LIN {X 0,Y 100.665,Z 312.75,A -85,B 0,C 180,E1 -26589.863,E2 -26589.863} C_VEL
LIN {X 0,Y 100.701,Z 312.753,A -85,B 0,C 180,E1 -26595.772,E2 -26595.772} C_VEL
LIN {X 0,Y 100.661,Z 312.753,A -85,B 0,C 180,E1 -26601.099,E2 -26601.099} C_VEL
LIN {X 0,Y 100.673,Z 312.753,A -85,B 0,C 180,E1 -26606.886,E2 -26606.886} C_VEL
LIN {X 0,Y 100.759,Z 312.744,A -85,B 0,C 180,E1 -26615.283,E2 -26615.283} C_VEL
LIN {X 0,Y 100.778,Z 312.74,A -85,B 0,C 180,E1 -26619.616,E2 -26619.616} C_VEL
LIN {X 0,Y 101.104,Z 312.698,A -85,B 0,C 180,E1 -26627.985,E2 -26627.985} C_VEL
LIN {X 0,Y 101.211,Z 312.69,A -85,B 0,C 180,E1 -26632.038,E2 -26632.038} C_VEL
LIN {X 0,Y 101.814,Z 312.615,A -85,B 0,C 180,E1 -26640.02,E2 -26640.02} C_VEL
LIN {X 0,Y 101.213,Z 312.689,A -85,B 0,C 180,E1 -26648.003,E2 -26648.003} C_VEL
LIN {X 0,Y 101.044,Z 312.702,A -85,B 0,C 180,E1 -26653.189,E2 -26653.189} C_VEL
LIN {X 0,Y 100.771,Z 312.742,A -85,B 0,C 180,E1 -26660.429,E2 -26660.429} C_VEL
LIN {X 0,Y 100.702,Z 312.75,A -85,B 0,C 180,E1 -26664.887,E2 -26664.887} C_VEL
LIN {X 0,Y 100.687,Z 312.75,A -85,B 0,C 180,E1 -26673.125,E2 -26673.125} C_VEL
LIN {X 0,Y 100.643,Z 312.753,A -85,B 0,C 180,E1 -26679.824,E2 -26679.824} C_VEL
LIN {X 0,Y 100.652,Z 312.76,A -85,B 0,C 180,E1 -26685.724,E2 -26685.724} C_VEL
LIN {X 0,Y 100.635,Z 312.757,A -85,B 0,C 180,E1 -26691.068,E2 -26691.068} C_VEL
LIN {X 0,Y 100.747,Z 312.743,A -85,B 0,C 180,E1 -26696.867,E2 -26696.867} C_VEL
LIN {X 0,Y 100.816,Z 312.737,A -85,B 0,C 180,E1 -26700.8,E2 -26700.8} C_VEL
LIN {X 0,Y 100.943,Z 312.723,A -85,B 0,C 180,E1 -26705.316,E2 -26705.316} C_VEL
LIN {X 0,Y 101.451,Z 312.659,A -85,B 0,C 180,E1 -26718.012,E2 -26718.012} C_VEL
LIN {X 0,Y 102.379,Z 312.611,A -85,B 0,C 180,E1 -26720.25,E2 -26720.25} C_VEL
LIN {X 0,Y 104.384,Z 336.262,A -85,B 0,C 180,E1 -26723.361,E2 -26723.361} C_VEL
LIN {X 0,Y 106.398,Z 352.42,A -85,B 0,C 180,E1 -26725.335,E2 -26725.335} C_VEL
LIN {X 0,Y 107.925,Z 383.014,A -85,B 0,C 180,E1 -26729.89,E2 -26729.89} C_VEL
LIN {X 0,Y 108.387,Z 393.278,A -85,B 0,C 180,E1 -26731.864,E2 -26731.864} C_VEL
LIN {X 0,Y 108.985,Z 404.094,A -85,B 0,C 180,E1 -26734.63,E2 -26734.63} C_VEL
LIN {X 0,Y 109.704,Z 414.44,A -85,B 0,C 180,E1 -26738.136,E2 -26738.136} C_VEL
LIN {X 0,Y 109.906,Z 418.538,A -85,B 0,C 180,E1 -26739.991,E2 -26739.991} C_VEL
LIN {X 0,Y 109.314,Z 424.896,A -85,B 0,C 180,E1 -26744.01,E2 -26744.01} C_VEL
LIN {X 0,Y 109.51,Z 433.596,A -85,B 0,C 180,E1 -26750.675,E2 -26750.675} C_VEL
LIN {X 0,Y 112.549,Z 441.833,A -85,B 0,C 180,E1 -26758.135,E2 -26758.135} C_VEL
LIN {X 0,Y 116.222,Z 446.661,A -85,B 0,C 180,E1 -26762.979,E2 -26762.979} C_VEL
LIN {X 0,Y 121.104,Z 450.868,A -85,B 0,C 180,E1 -26767.548,E2 -26767.548} C_VEL
LIN {X 0,Y 127.149,Z 454.377,A -85,B 0,C 180,E1 -26771.557,E2 -26771.557} C_VEL
LIN {X 0,Y 131.686,Z 456.416,A -85,B 0,C 180,E1 -26773.938,E2 -26773.938} C_VEL
LIN {X 0,Y 136.655,Z 458.059,A -85,B 0,C 180,E1 -26776.061,E2 -26776.061} C_VEL
LIN {X 0,Y 129.507,Z 454.575,A -85,B 0,C 180,E1 -26779.349,E2 -26779.349} C_VEL
LIN {X 0,Y 122.955,Z 450.261,A -85,B 0,C 180,E1 -26783.1,E2 -26783.1} C_VEL
LIN {X 0,Y 117.303,Z 444.969,A -85,B 0,C 180,E1 -26787.351,E2 -26787.351} C_VEL
LIN {X 0,Y 112.243,Z 437.819,A -85,B 0,C 180,E1 -26792.944,E2 -26792.944} C_VEL
LIN {X 0,Y 108.802,Z 428.944,A -85,B 0,C 180,E1 -26799.172,E2 -26799.172} C_VEL
LIN {X 0,Y 107.58,Z 421.613,A -85,B 0,C 180,E1 -26803.862,E2 -26803.862} C_VEL
LIN {X 0,Y 107.219,Z 414.624,A -85,B 0,C 180,E1 -26807.681,E2 -26807.681} C_VEL
LIN {X 0,Y 107.195,Z 406.282,A -85,B 0,C 180,E1 -26811.497,E2 -26811.497} C_VEL
LIN {X 0,Y 107.087,Z 396.993,A -85,B 0,C 180,E1 -26814.804,E2 -26814.804} C_VEL
LIN {X 0,Y 106.94,Z 388.426,A -85,B 0,C 180,E1 -26817.156,E2 -26817.156} C_VEL
LIN {X 0,Y 106.923,Z 378.584,A -85,B 0,C 180,E1 -26819.275,E2 -26819.275} C_VEL
LIN {X 0,Y 106.708,Z 365.006,A -85,B 0,C 180,E1 -26821.514,E2 -26821.514} C_VEL
LIN {X 0,Y 106.169,Z 353.16,A -85,B 0,C 180,E1 -26823.272,E2 -26823.272} C_VEL
LIN {X 0,Y 105.327,Z 347.436,A -85,B 0,C 180,E1 -26823.931,E2 -26823.931} C_VEL
LIN {X 0,Y 99.604,Z 328.593,A -85,B 0,C 180,E1 -26825.273,E2 -26825.273} C_VEL
LIN {X 0,Y 98.786,Z 322.861,A -85,B 0,C 180,E1 -26825.965,E2 -26825.965} C_VEL
LIN {X 0,Y 97.433,Z 313.16,A -85,B 0,C 180,E1 -26827.229,E2 -26827.229} C_VEL
LIN {X 0,Y 94.53,Z 313.52,A -85,B 0,C 180,E1 -26834.845,E2 -26834.845} C_VEL
LIN {X 0,Y 93.661,Z 313.629,A -85,B 0,C 180,E1 -26845.77,E2 -26845.77} C_VEL
LIN {X 0,Y 93.57,Z 313.64,A -85,B 0,C 180,E1 -26854.277,E2 -26854.277} C_VEL
LIN {X 0,Y 93.507,Z 313.646,A -85,B 0,C 180,E1 -26862.534,E2 -26862.534} C_VEL
LIN {X 0,Y 93.506,Z 313.642,A -85,B 0,C 180,E1 -26868.693,E2 -26868.693} C_VEL
LIN {X 0,Y 93.556,Z 313.642,A -85,B 0,C 180,E1 -26875.68,E2 -26875.68} C_VEL
LIN {X 0,Y 93.637,Z 313.633,A -85,B 0,C 180,E1 -26884.19,E2 -26884.19} C_VEL
LIN {X 0,Y 93.657,Z 313.623,A -85,B 0,C 180,E1 -26887.956,E2 -26887.956} C_VEL
LIN {X 0,Y 94.038,Z 313.575,A -85,B 0,C 180,E1 -26897.036,E2 -26897.036} C_VEL
LIN {X 0,Y 94.149,Z 313.57,A -85,B 0,C 180,E1 -26901.407,E2 -26901.407} C_VEL
LIN {X 0,Y 94.76,Z 313.495,A -85,B 0,C 180,E1 -26909.993,E2 -26909.993} C_VEL
LIN {X 0,Y 94.145,Z 313.571,A -85,B 0,C 180,E1 -26918.579,E2 -26918.579} C_VEL
LIN {X 0,Y 93.987,Z 313.581,A -85,B 0,C 180,E1 -26923.673,E2 -26923.673} C_VEL
LIN {X 0,Y 93.648,Z 313.624,A -85,B 0,C 180,E1 -26932.031,E2 -26932.031} C_VEL
LIN {X 0,Y 93.582,Z 313.641,A -85,B 0,C 180,E1 -26936.773,E2 -26936.773} C_VEL
LIN {X 0,Y 93.574,Z 313.639,A -85,B 0,C 180,E1 -26944.336,E2 -26944.336} C_VEL
LIN {X 0,Y 93.597,Z 313.635,A -85,B 0,C 180,E1 -26952.505,E2 -26952.505} C_VEL
LIN {X 0,Y 93.594,Z 313.632,A -85,B 0,C 180,E1 -26958.656,E2 -26958.656} C_VEL
LIN {X 0,Y 93.58,Z 313.639,A -85,B 0,C 180,E1 -26965.687,E2 -26965.687} C_VEL
LIN {X 0,Y 93.641,Z 313.632,A -85,B 0,C 180,E1 -26974.223,E2 -26974.223} C_VEL
LIN {X 0,Y 93.658,Z 313.623,A -85,B 0,C 180,E1 -26977.988,E2 -26977.988} C_VEL
LIN {X 0,Y 93.996,Z 313.581,A -85,B 0,C 180,E1 -26987.061,E2 -26987.061} C_VEL
LIN {X 0,Y 94.141,Z 313.571,A -85,B 0,C 180,E1 -26991.435,E2 -26991.435} C_VEL
LIN {X 0,Y 94.743,Z 313.496,A -85,B 0,C 180,E1 -27000.021,E2 -27000.021} C_VEL
LIN {X 0,Y 94.143,Z 313.571,A -85,B 0,C 180,E1 -27008.608,E2 -27008.608} C_VEL
LIN {X 0,Y 93.952,Z 313.585,A -85,B 0,C 180,E1 -27013.514,E2 -27013.514} C_VEL
LIN {X 0,Y 93.634,Z 313.625,A -85,B 0,C 180,E1 -27022.064,E2 -27022.064} C_VEL
LIN {X 0,Y 93.55,Z 313.644,A -85,B 0,C 180,E1 -27026.815,E2 -27026.815} C_VEL
LIN {X 0,Y 93.586,Z 313.638,A -85,B 0,C 180,E1 -27034.318,E2 -27034.318} C_VEL
LIN {X 0,Y 93.538,Z 313.643,A -85,B 0,C 180,E1 -27042.575,E2 -27042.575} C_VEL
LIN {X 0,Y 93.544,Z 313.638,A -85,B 0,C 180,E1 -27048.733,E2 -27048.733} C_VEL
LIN {X 0,Y 93.626,Z 313.634,A -85,B 0,C 180,E1 -27055.694,E2 -27055.694} C_VEL
LIN {X 0,Y 93.787,Z 313.615,A -85,B 0,C 180,E1 -27063.29,E2 -27063.29} C_VEL
LIN {X 0,Y 93.638,Z 313.628,A -85,B 0,C 180,E1 -27067.967,E2 -27067.967} C_VEL
LIN {X 0,Y 94.083,Z 313.573,A -85,B 0,C 180,E1 -27077.058,E2 -27077.058} C_VEL
LIN {X 0,Y 96.014,Z 313.336,A -85,B 0,C 180,E1 -27082.099,E2 -27082.099} C_VEL
LIN {X 0,Y 98.175,Z 336.207,A -85,B 0,C 180,E1 -27085.298,E2 -27085.298} C_VEL
LIN {X 0,Y 100.242,Z 351.555,A -85,B 0,C 180,E1 -27087.244,E2 -27087.244} C_VEL
LIN {X 0,Y 102.166,Z 383.219,A -85,B 0,C 180,E1 -27092.224,E2 -27092.224} C_VEL
LIN {X 0,Y 102.668,Z 392.712,A -85,B 0,C 180,E1 -27094.178,E2 -27094.178} C_VEL
LIN {X 0,Y 103.409,Z 402.496,A -85,B 0,C 180,E1 -27096.837,E2 -27096.837} C_VEL
LIN {X 0,Y 104.274,Z 412.028,A -85,B 0,C 180,E1 -27100.197,E2 -27100.197} C_VEL
LIN {X 0,Y 104.461,Z 415.18,A -85,B 0,C 180,E1 -27101.651,E2 -27101.651} C_VEL
LIN {X 0,Y 103.914,Z 421.503,A -85,B 0,C 180,E1 -27105.703,E2 -27105.703} C_VEL
LIN {X 0,Y 104.221,Z 429.208,A -85,B 0,C 180,E1 -27111.777,E2 -27111.777} C_VEL
LIN {X 0,Y 106.678,Z 437.042,A -85,B 0,C 180,E1 -27118.645,E2 -27118.645} C_VEL
LIN {X 0,Y 112.583,Z 444.916,A -85,B 0,C 180,E1 -27126.38,E2 -27126.38} C_VEL
LIN {X 0,Y 118.015,Z 449.228,A -85,B 0,C 180,E1 -27130.932,E2 -27130.932} C_VEL
LIN {X 0,Y 126.967,Z 453.986,A -85,B 0,C 180,E1 -27136.027,E2 -27136.027} C_VEL
LIN {X 0,Y 117.676,Z 447.719,A -85,B 0,C 180,E1 -27141.144,E2 -27141.144} C_VEL
LIN {X 0,Y 111.038,Z 440.965,A -85,B 0,C 180,E1 -27146.351,E2 -27146.351} C_VEL
LIN {X 0,Y 106.067,Z 432.912,A -85,B 0,C 180,E1 -27152.346,E2 -27152.346} C_VEL
LIN {X 0,Y 103.591,Z 426.177,A -85,B 0,C 180,E1 -27157.019,E2 -27157.019} C_VEL
LIN {X 0,Y 102.021,Z 416.844,A -85,B 0,C 180,E1 -27162.956,E2 -27162.956} C_VEL
LIN {X 0,Y 101.631,Z 408.488,A -85,B 0,C 180,E1 -27167.449,E2 -27167.449} C_VEL
LIN {X 0,Y 101.499,Z 400.712,A -85,B 0,C 180,E1 -27170.737,E2 -27170.737} C_VEL
LIN {X 0,Y 101.294,Z 390.735,A -85,B 0,C 180,E1 -27174.007,E2 -27174.007} C_VEL
LIN {X 0,Y 101.084,Z 379.599,A -85,B 0,C 180,E1 -27176.723,E2 -27176.723} C_VEL
LIN {X 0,Y 100.766,Z 365.78,A -85,B 0,C 180,E1 -27179.273,E2 -27179.273} C_VEL
LIN {X 0,Y 98.786,Z 322.861,A -85,B 0,C 180,E1 -27185.965,E2 -27185.965} C_VEL
LIN {X 0,Y 98.291,Z 320.434,A -85,B 0,C 180,E1 -27186.595,E2 -27186.595} C_VEL
LIN {X 0,Y 96.85,Z 317.92,A -85,B 0,C 180,E1 -27187.917,E2 -27187.917} C_VEL
LIN {X 0,Y 94.432,Z 315.841,A -85,B 0,C 180,E1 -27190.08,E2 -27190.08} C_VEL
LIN {X 0,Y 91.311,Z 314.68,A -85,B 0,C 180,E1 -27193.245,E2 -27193.245} C_VEL
LIN {X 0,Y 87.725,Z 314.403,A -85,B 0,C 180,E1 -27198.434,E2 -27198.434} C_VEL
LIN {X 0,Y 86.632,Z 314.494,A -85,B 0,C 180,E1 -27202.725,E2 -27202.725} C_VEL
LIN {X 0,Y 86.461,Z 314.525,A -85,B 0,C 180,E1 -27209.161,E2 -27209.161} C_VEL
LIN {X 0,Y 86.487,Z 314.524,A -85,B 0,C 180,E1 -27215.636,E2 -27215.636} C_VEL
LIN {X 0,Y 86.451,Z 314.526,A -85,B 0,C 180,E1 -27222.965,E2 -27222.965} C_VEL
LIN {X 0,Y 86.429,Z 314.522,A -85,B 0,C 180,E1 -27229.409,E2 -27229.409} C_VEL
LIN {X 0,Y 86.499,Z 314.521,A -85,B 0,C 180,E1 -27235.328,E2 -27235.328} C_VEL
LIN {X 0,Y 86.552,Z 314.517,A -85,B 0,C 180,E1 -27243.22,E2 -27243.22} C_VEL
LIN {X 0,Y 86.609,Z 314.508,A -85,B 0,C 180,E1 -27251.052,E2 -27251.052} C_VEL
LIN {X 0,Y 86.895,Z 314.464,A -85,B 0,C 180,E1 -27255.95,E2 -27255.95} C_VEL
LIN {X 0,Y 87.057,Z 314.453,A -85,B 0,C 180,E1 -27260.701,E2 -27260.701} C_VEL
LIN {X 0,Y 87.687,Z 314.376,A -85,B 0,C 180,E1 -27269.992,E2 -27269.992} C_VEL
LIN {X 0,Y 87.053,Z 314.453,A -85,B 0,C 180,E1 -27279.284,E2 -27279.284} C_VEL
LIN {X 0,Y 86.89,Z 314.465,A -85,B 0,C 180,E1 -27284.035,E2 -27284.035} C_VEL
LIN {X 0,Y 86.601,Z 314.509,A -85,B 0,C 180,E1 -27288.934,E2 -27288.934} C_VEL
LIN {X 0,Y 86.544,Z 314.518,A -85,B 0,C 180,E1 -27296.771,E2 -27296.771} C_VEL
LIN {X 0,Y 86.499,Z 314.523,A -85,B 0,C 180,E1 -27305.704,E2 -27305.704} C_VEL
LIN {X 0,Y 86.524,Z 314.517,A -85,B 0,C 180,E1 -27313.065,E2 -27313.065} C_VEL
LIN {X 0,Y 86.519,Z 314.511,A -85,B 0,C 180,E1 -27319.504,E2 -27319.504} C_VEL
LIN {X 0,Y 86.528,Z 314.518,A -85,B 0,C 180,E1 -27325.381,E2 -27325.381} C_VEL
LIN {X 0,Y 86.556,Z 314.516,A -85,B 0,C 180,E1 -27333.254,E2 -27333.254} C_VEL
LIN {X 0,Y 86.595,Z 314.51,A -85,B 0,C 180,E1 -27341.082,E2 -27341.082} C_VEL
LIN {X 0,Y 86.859,Z 314.469,A -85,B 0,C 180,E1 -27346.119,E2 -27346.119} C_VEL
LIN {X 0,Y 87.044,Z 314.455,A -85,B 0,C 180,E1 -27350.731,E2 -27350.731} C_VEL
LIN {X 0,Y 87.673,Z 314.377,A -85,B 0,C 180,E1 -27360.023,E2 -27360.023} C_VEL
LIN {X 0,Y 87.049,Z 314.454,A -85,B 0,C 180,E1 -27369.315,E2 -27369.315} C_VEL
LIN {X 0,Y 86.854,Z 314.47,A -85,B 0,C 180,E1 -27374.072,E2 -27374.072} C_VEL
LIN {X 0,Y 86.587,Z 314.511,A -85,B 0,C 180,E1 -27378.969,E2 -27378.969} C_VEL
LIN {X 0,Y 86.525,Z 314.519,A -85,B 0,C 180,E1 -27386.706,E2 -27386.706} C_VEL
LIN {X 0,Y 86.507,Z 314.523,A -85,B 0,C 180,E1 -27395.681,E2 -27395.681} C_VEL
LIN {X 0,Y 86.462,Z 314.525,A -85,B 0,C 180,E1 -27402.995,E2 -27402.995} C_VEL
LIN {X 0,Y 86.468,Z 314.518,A -85,B 0,C 180,E1 -27409.452,E2 -27409.452} C_VEL
LIN {X 0,Y 86.566,Z 314.514,A -85,B 0,C 180,E1 -27415.378,E2 -27415.378} C_VEL
LIN {X 0,Y 86.718,Z 314.495,A -85,B 0,C 180,E1 -27423.105,E2 -27423.105} C_VEL
LIN {X 0,Y 86.501,Z 314.523,A -85,B 0,C 180,E1 -27431.044,E2 -27431.044} C_VEL
LIN {X 0,Y 88.127,Z 314.318,A -85,B 0,C 180,E1 -27440.83,E2 -27440.83} C_VEL
LIN {X 0,Y 89.757,Z 314.11,A -85,B 0,C 180,E1 -27444.25,E2 -27444.25} C_VEL
LIN {X 0,Y 92.272,Z 337.546,A -85,B 0,C 180,E1 -27447.687,E2 -27447.687} C_VEL
LIN {X 0,Y 94.26,Z 351.179,A -85,B 0,C 180,E1 -27449.488,E2 -27449.488} C_VEL
LIN {X 0,Y 96.686,Z 382.911,A -85,B 0,C 180,E1 -27454.828,E2 -27454.828} C_VEL
LIN {X 0,Y 97.469,Z 393.635,A -85,B 0,C 180,E1 -27457.256,E2 -27457.256} C_VEL
LIN {X 0,Y 98.39,Z 403.722,A -85,B 0,C 180,E1 -27460.294,E2 -27460.294} C_VEL
LIN {X 0,Y 99.138,Z 410.816,A -85,B 0,C 180,E1 -27463.058,E2 -27463.058} C_VEL
LIN {X 0,Y 98.946,Z 414.824,A -85,B 0,C 180,E1 -27465.418,E2 -27465.418} C_VEL
LIN {X 0,Y 98.986,Z 423.465,A -85,B 0,C 180,E1 -27472.001,E2 -27472.001} C_VEL
LIN {X 0,Y 100.588,Z 430.572,A -85,B 0,C 180,E1 -27478.147,E2 -27478.147} C_VEL
LIN {X 0,Y 104.715,Z 437.975,A -85,B 0,C 180,E1 -27485.018,E2 -27485.018} C_VEL
LIN {X 0,Y 111.315,Z 444.509,A -85,B 0,C 180,E1 -27491.531,E2 -27491.531} C_VEL
LIN {X 0,Y 117.69,Z 448.827,A -85,B 0,C 180,E1 -27495.781,E2 -27495.781} C_VEL
LIN {X 0,Y 117.158,Z 448.434,A -85,B 0,C 180,E1 -27496.358,E2 -27496.358} C_VEL
LIN {X 0,Y 108.566,Z 440.736,A -85,B 0,C 180,E1 -27502.028,E2 -27502.028} C_VEL
LIN {X 0,Y 104.228,Z 435.253,A -85,B 0,C 180,E1 -27506.179,E2 -27506.179} C_VEL
LIN {X 0,Y 100.153,Z 427.508,A -85,B 0,C 180,E1 -27511.706,E2 -27511.706} C_VEL
LIN {X 0,Y 97.873,Z 420.23,A -85,B 0,C 180,E1 -27516.717,E2 -27516.717} C_VEL
LIN {X 0,Y 96.686,Z 410.847,A -85,B 0,C 180,E1 -27522.476,E2 -27522.476} C_VEL
LIN {X 0,Y 96.23,Z 401.198,A -85,B 0,C 180,E1 -27527.323,E2 -27527.323} C_VEL
LIN {X 0,Y 95.904,Z 392.21,A -85,B 0,C 180,E1 -27530.645,E2 -27530.645} C_VEL
LIN {X 0,Y 95.59,Z 380.07,A -85,B 0,C 180,E1 -27533.912,E2 -27533.912} C_VEL
LIN {X 0,Y 95.058,Z 365.316,A -85,B 0,C 180,E1 -27536.8,E2 -27536.8} C_VEL
LIN {X 0,Y 92.405,Z 320.941,A -85,B 0,C 180,E1 -27544.248,E2 -27544.248} C_VEL
LIN {X 0,Y 91.254,Z 313.926,A -85,B 0,C 180,E1 -27545.122,E2 -27545.122} C_VEL
LIN {X 0,Y 89.146,Z 314.195,A -85,B 0,C 180,E1 -27549.048,E2 -27549.048} C_VEL
LIN {X 0,Y 86.632,Z 314.494,A -85,B 0,C 180,E1 -27562.725,E2 -27562.725} C_VEL
LIN {X 0,Y 86.231,Z 314.554,A -85,B 0,C 180,E1 -27565.314,E2 -27565.314} C_VEL
LIN {X 0,Y 84.74,Z 314.743,A -85,B 0,C 180,E1 -27569.154,E2 -27569.154} C_VEL
LIN {X 0,Y 79.479,Z 315.389,A -85,B 0,C 180,E1 -27581.333,E2 -27581.333} C_VEL
LIN {X 0,Y 79.318,Z 315.412,A -85,B 0,C 180,E1 -27584.259,E2 -27584.259} C_VEL
LIN {X 0,Y 79.357,Z 315.411,A -85,B 0,C 180,E1 -27592.803,E2 -27592.803} C_VEL
LIN {X 0,Y 79.449,Z 315.4,A -85,B 0,C 180,E1 -27602.14,E2 -27602.14} C_VEL
LIN {X 0,Y 79.478,Z 315.392,A -85,B 0,C 180,E1 -27609.277,E2 -27609.277} C_VEL
LIN {X 0,Y 79.79,Z 315.35,A -85,B 0,C 180,E1 -27615.557,E2 -27615.557} C_VEL
LIN {X 0,Y 79.937,Z 315.339,A -85,B 0,C 180,E1 -27619.864,E2 -27619.864} C_VEL
LIN {X 0,Y 80.614,Z 315.257,A -85,B 0,C 180,E1 -27629.992,E2 -27629.992} C_VEL
LIN {X 0,Y 79.933,Z 315.34,A -85,B 0,C 180,E1 -27640.119,E2 -27640.119} C_VEL
LIN {X 0,Y 79.702,Z 315.364,A -85,B 0,C 180,E1 -27645.33,E2 -27645.33} C_VEL
LIN {X 0,Y 79.469,Z 315.393,A -85,B 0,C 180,E1 -27650.707,E2 -27650.707} C_VEL
LIN {X 0,Y 79.443,Z 315.401,A -85,B 0,C 180,E1 -27657.852,E2 -27657.852} C_VEL
LIN {X 0,Y 79.415,Z 315.404,A -85,B 0,C 180,E1 -27667.251,E2 -27667.251} C_VEL
LIN {X 0,Y 79.432,Z 315.404,A -85,B 0,C 180,E1 -27675.046,E2 -27675.046} C_VEL
LIN {X 0,Y 79.419,Z 315.403,A -85,B 0,C 180,E1 -27682.775,E2 -27682.775} C_VEL
LIN {X 0,Y 79.454,Z 315.401,A -85,B 0,C 180,E1 -27692.175,E2 -27692.175} C_VEL
LIN {X 0,Y 79.472,Z 315.393,A -85,B 0,C 180,E1 -27699.313,E2 -27699.313} C_VEL
LIN {X 0,Y 79.761,Z 315.354,A -85,B 0,C 180,E1 -27705.716,E2 -27705.716} C_VEL
LIN {X 0,Y 79.922,Z 315.341,A -85,B 0,C 180,E1 -27709.897,E2 -27709.897} C_VEL
LIN {X 0,Y 80.603,Z 315.257,A -85,B 0,C 180,E1 -27720.025,E2 -27720.025} C_VEL
LIN {X 0,Y 79.925,Z 315.341,A -85,B 0,C 180,E1 -27730.154,E2 -27730.154} C_VEL
LIN {X 0,Y 79.682,Z 315.367,A -85,B 0,C 180,E1 -27735.369,E2 -27735.369} C_VEL
LIN {X 0,Y 79.459,Z 315.394,A -85,B 0,C 180,E1 -27740.745,E2 -27740.745} C_VEL
LIN {X 0,Y 79.421,Z 315.404,A -85,B 0,C 180,E1 -27747.781,E2 -27747.781} C_VEL
LIN {X 0,Y 79.345,Z 315.405,A -85,B 0,C 180,E1 -27752.131,E2 -27752.131} C_VEL
LIN {X 0,Y 79.37,Z 315.407,A -85,B 0,C 180,E1 -27758.334,E2 -27758.334} C_VEL
LIN {X 0,Y 79.395,Z 315.408,A -85,B 0,C 180,E1 -27765.118,E2 -27765.118} C_VEL
LIN {X 0,Y 79.409,Z 315.405,A -85,B 0,C 180,E1 -27772.839,E2 -27772.839} C_VEL
LIN {X 0,Y 79.621,Z 315.379,A -85,B 0,C 180,E1 -27782.016,E2 -27782.016} C_VEL
LIN {X 0,Y 79.45,Z 315.398,A -85,B 0,C 180,E1 -27789.288,E2 -27789.288} C_VEL
LIN {X 0,Y 80.661,Z 315.247,A -85,B 0,C 180,E1 -27799.973,E2 -27799.973} C_VEL
LIN {X 0,Y 83.808,Z 314.862,A -85,B 0,C 180,E1 -27806.885,E2 -27806.885} C_VEL
LIN {X 0,Y 86.75,Z 338.79,A -85,B 0,C 180,E1 -27810.516,E2 -27810.516} C_VEL
LIN {X 0,Y 88.662,Z 351.424,A -85,B 0,C 180,E1 -27812.279,E2 -27812.279} C_VEL
LIN {X 0,Y 91.375,Z 381.665,A -85,B 0,C 180,E1 -27817.604,E2 -27817.604} C_VEL
LIN {X 0,Y 92.214,Z 391.506,A -85,B 0,C 180,E1 -27819.881,E2 -27819.881} C_VEL
LIN {X 0,Y 93.145,Z 400.297,A -85,B 0,C 180,E1 -27822.536,E2 -27822.536} C_VEL
LIN {X 0,Y 94.053,Z 407.162,A -85,B 0,C 180,E1 -27825.168,E2 -27825.168} C_VEL
LIN {X 0,Y 94.054,Z 410.92,A -85,B 0,C 180,E1 -27827.398,E2 -27827.398} C_VEL
LIN {X 0,Y 94.378,Z 420.929,A -85,B 0,C 180,E1 -27835.213,E2 -27835.213} C_VEL
LIN {X 0,Y 97.286,Z 429.392,A -85,B 0,C 180,E1 -27842.814,E2 -27842.814} C_VEL
LIN {X 0,Y 101.408,Z 435.563,A -85,B 0,C 180,E1 -27848.597,E2 -27848.597} C_VEL
LIN {X 0,Y 108.867,Z 442.529,A -85,B 0,C 180,E1 -27855.252,E2 -27855.252} C_VEL
LIN {X 0,Y 107.666,Z 441.279,A -85,B 0,C 180,E1 -27856.965,E2 -27856.965} C_VEL
LIN {X 0,Y 100.944,Z 433.671,A -85,B 0,C 180,E1 -27862.446,E2 -27862.446} C_VEL
LIN {X 0,Y 96.984,Z 427.318,A -85,B 0,C 180,E1 -27867.056,E2 -27867.056} C_VEL
LIN {X 0,Y 93.114,Z 416.885,A -85,B 0,C 180,E1 -27874.282,E2 -27874.282} C_VEL
LIN {X 0,Y 91.723,Z 407.604,A -85,B 0,C 180,E1 -27880.1,E2 -27880.1} C_VEL
LIN {X 0,Y 91.279,Z 399.872,A -85,B 0,C 180,E1 -27884.112,E2 -27884.112} C_VEL
LIN {X 0,Y 90.791,Z 390.821,A -85,B 0,C 180,E1 -27887.687,E2 -27887.687} C_VEL
LIN {X 0,Y 90.263,Z 379.883,A -85,B 0,C 180,E1 -27890.878,E2 -27890.878} C_VEL
LIN {X 0,Y 89.58,Z 365.368,A -85,B 0,C 180,E1 -27893.926,E2 -27893.926} C_VEL
LIN {X 0,Y 86.423,Z 321.198,A -85,B 0,C 180,E1 -27901.797,E2 -27901.797} C_VEL
LIN {X 0,Y 85.244,Z 314.674,A -85,B 0,C 180,E1 -27902.708,E2 -27902.708} C_VEL
LIN {X 0,Y 83.804,Z 314.852,A -85,B 0,C 180,E1 -27904.786,E2 -27904.786} C_VEL
LIN {X 0,Y 79.565,Z 315.373,A -85,B 0,C 180,E1 -27922.535,E2 -27922.535} C_VEL
LIN {X 0,Y 79.471,Z 315.398,A -85,B 0,C 180,E1 -27927.812,E2 -27927.812} C_VEL
LIN {X 0,Y 79.367,Z 315.41,A -85,B 0,C 180,E1 -27937.147,E2 -27937.147} C_VEL
LIN {X 0,Y 79.318,Z 315.412,A -85,B 0,C 180,E1 -27944.259,E2 -27944.259} C_VEL
LIN {X 0,Y 79.152,Z 315.453,A -85,B 0,C 180,E1 -27947.087,E2 -27947.087} C_VEL
LIN {X 0,Y 77.932,Z 315.621,A -85,B 0,C 180,E1 -27951.302,E2 -27951.302} C_VEL
LIN {X 0,Y 74.763,Z 316.01,A -85,B 0,C 180,E1 -27958.483,E2 -27958.483} C_VEL
LIN {X 0,Y 72.708,Z 316.241,A -85,B 0,C 180,E1 -27964.68,E2 -27964.68} C_VEL
LIN {X 0,Y 72.339,Z 316.273,A -85,B 0,C 180,E1 -27967.914,E2 -27967.914} C_VEL
LIN {X 0,Y 72.686,Z 316.236,A -85,B 0,C 180,E1 -27975.095,E2 -27975.095} C_VEL
LIN {X 0,Y 72.827,Z 316.223,A -85,B 0,C 180,E1 -27978.862,E2 -27978.862} C_VEL
LIN {X 0,Y 73.54,Z 316.138,A -85,B 0,C 180,E1 -27989.991,E2 -27989.991} C_VEL
LIN {X 0,Y 72.822,Z 316.224,A -85,B 0,C 180,E1 -28001.119,E2 -28001.119} C_VEL
LIN {X 0,Y 72.532,Z 316.262,A -85,B 0,C 180,E1 -28006.889,E2 -28006.889} C_VEL
LIN {X 0,Y 72.352,Z 316.276,A -85,B 0,C 180,E1 -28012.854,E2 -28012.854} C_VEL
LIN {X 0,Y 72.337,Z 316.283,A -85,B 0,C 180,E1 -28019.089,E2 -28019.089} C_VEL
LIN {X 0,Y 72.3,Z 316.292,A -85,B 0,C 180,E1 -28025.666,E2 -28025.666} C_VEL
LIN {X 0,Y 72.276,Z 316.291,A -85,B 0,C 180,E1 -28032.882,E2 -28032.882} C_VEL
LIN {X 0,Y 72.326,Z 316.282,A -85,B 0,C 180,E1 -28041.005,E2 -28041.005} C_VEL
LIN {X 0,Y 72.305,Z 316.291,A -85,B 0,C 180,E1 -28044.361,E2 -28044.361} C_VEL
LIN {X 0,Y 72.363,Z 316.281,A -85,B 0,C 180,E1 -28050.982,E2 -28050.982} C_VEL
LIN {X 0,Y 72.359,Z 316.275,A -85,B 0,C 180,E1 -28057.17,E2 -28057.17} C_VEL
LIN {X 0,Y 72.658,Z 316.239,A -85,B 0,C 180,E1 -28065.261,E2 -28065.261} C_VEL
LIN {X 0,Y 72.809,Z 316.225,A -85,B 0,C 180,E1 -28068.898,E2 -28068.898} C_VEL
LIN {X 0,Y 73.531,Z 316.138,A -85,B 0,C 180,E1 -28080.028,E2 -28080.028} C_VEL
LIN {X 0,Y 72.818,Z 316.223,A -85,B 0,C 180,E1 -28091.157,E2 -28091.157} C_VEL
LIN {X 0,Y 72.497,Z 316.266,A -85,B 0,C 180,E1 -28096.936,E2 -28096.936} C_VEL
LIN {X 0,Y 72.344,Z 316.276,A -85,B 0,C 180,E1 -28102.895,E2 -28102.895} C_VEL
LIN {X 0,Y 72.315,Z 316.286,A -85,B 0,C 180,E1 -28109.103,E2 -28109.103} C_VEL
LIN {X 0,Y 72.289,Z 316.293,A -85,B 0,C 180,E1 -28115.717,E2 -28115.717} C_VEL
LIN {X 0,Y 72.254,Z 316.294,A -85,B 0,C 180,E1 -28122.947,E2 -28122.947} C_VEL
LIN {X 0,Y 72.311,Z 316.284,A -85,B 0,C 180,E1 -28131.075,E2 -28131.075} C_VEL
LIN {X 0,Y 72.483,Z 316.265,A -85,B 0,C 180,E1 -28140.818,E2 -28140.818} C_VEL
LIN {X 0,Y 72.401,Z 316.271,A -85,B 0,C 180,E1 -28147.163,E2 -28147.163} C_VEL
LIN {X 0,Y 75.084,Z 315.939,A -85,B 0,C 180,E1 -28164.638,E2 -28164.638} C_VEL
LIN {X 0,Y 78.13,Z 315.681,A -85,B 0,C 180,E1 -28169.929,E2 -28169.929} C_VEL
LIN {X 0,Y 81.078,Z 337.742,A -85,B 0,C 180,E1 -28173.425,E2 -28173.425} C_VEL
LIN {X 0,Y 83.185,Z 350.295,A -85,B 0,C 180,E1 -28175.189,E2 -28175.189} C_VEL
LIN {X 0,Y 86.499,Z 381.584,A -85,B 0,C 180,E1 -28180.986,E2 -28180.986} C_VEL
LIN {X 0,Y 87.533,Z 391.069,A -85,B 0,C 180,E1 -28183.354,E2 -28183.354} C_VEL
LIN {X 0,Y 88.702,Z 399.582,A -85,B 0,C 180,E1 -28186.107,E2 -28186.107} C_VEL
LIN {X 0,Y 89.448,Z 405.007,A -85,B 0,C 180,E1 -28188.325,E2 -28188.325} C_VEL
LIN {X 0,Y 89.402,Z 412.899,A -85,B 0,C 180,E1 -28194.229,E2 -28194.229} C_VEL
LIN {X 0,Y 91.666,Z 422.307,A -85,B 0,C 180,E1 -28202.467,E2 -28202.467} C_VEL
LIN {X 0,Y 94.686,Z 428.096,A -85,B 0,C 180,E1 -28207.768,E2 -28207.768} C_VEL
LIN {X 0,Y 100.628,Z 435.105,A -85,B 0,C 180,E1 -28214.308,E2 -28214.308} C_VEL
LIN {X 0,Y 101.188,Z 435.575,A -85,B 0,C 180,E1 -28215.984,E2 -28215.984} C_VEL
LIN {X 0,Y 94.574,Z 426.864,A -85,B 0,C 180,E1 -28222.163,E2 -28222.163} C_VEL
LIN {X 0,Y 90.096,Z 417.876,A -85,B 0,C 180,E1 -28228.468,E2 -28228.468} C_VEL
LIN {X 0,Y 87.575,Z 407.545,A -85,B 0,C 180,E1 -28235.344,E2 -28235.344} C_VEL
LIN {X 0,Y 86.666,Z 398.916,A -85,B 0,C 180,E1 -28240.304,E2 -28240.304} C_VEL
LIN {X 0,Y 86.178,Z 391.955,A -85,B 0,C 180,E1 -28243.392,E2 -28243.392} C_VEL
LIN {X 0,Y 85.544,Z 381.767,A -85,B 0,C 180,E1 -28246.768,E2 -28246.768} C_VEL
LIN {X 0,Y 84.757,Z 368.523,A -85,B 0,C 180,E1 -28249.978,E2 -28249.978} C_VEL
LIN {X 0,Y 81.023,Z 327.502,A -85,B 0,C 180,E1 -28257.8,E2 -28257.8} C_VEL
LIN {X 0,Y 80.22,Z 319.12,A -85,B 0,C 180,E1 -28259.269,E2 -28259.269} C_VEL
LIN {X 0,Y 79.558,Z 315.388,A -85,B 0,C 180,E1 -28259.816,E2 -28259.816} C_VEL
LIN {X 0,Y 77.405,Z 315.65,A -85,B 0,C 180,E1 -28262.712,E2 -28262.712} C_VEL
LIN {X 0,Y 72.503,Z 316.257,A -85,B 0,C 180,E1 -28282.782,E2 -28282.782} C_VEL
LIN {X 0,Y 72.349,Z 316.283,A -85,B 0,C 180,E1 -28289.025,E2 -28289.025} C_VEL
LIN {X 0,Y 72.277,Z 316.294,A -85,B 0,C 180,E1 -28295.655,E2 -28295.655} C_VEL
LIN {X 0,Y 72.226,Z 316.297,A -85,B 0,C 180,E1 -28302.892,E2 -28302.892} C_VEL
LIN {X 0,Y 72.267,Z 316.289,A -85,B 0,C 180,E1 -28311.03,E2 -28311.03} C_VEL
LIN {X 0,Y 72.265,Z 316.296,A -85,B 0,C 180,E1 -28314.29,E2 -28314.29} C_VEL
LIN {X 0,Y 72.329,Z 316.284,A -85,B 0,C 180,E1 -28320.923,E2 -28320.923} C_VEL
LIN {X 0,Y 72.339,Z 316.273,A -85,B 0,C 180,E1 -28327.914,E2 -28327.914} C_VEL
LIN {X 0,Y 71.739,Z 316.361,A -85,B 0,C 180,E1 -28332.596,E2 -28332.596} C_VEL
LIN {X 0,Y 69.917,Z 316.588,A -85,B 0,C 180,E1 -28338.848,E2 -28338.848} C_VEL
LIN {X 0,Y 65.999,Z 317.061,A -85,B 0,C 180,E1 -28353.987,E2 -28353.987} C_VEL
LIN {X 0,Y 65.716,Z 317.103,A -85,B 0,C 180,E1 -28362.34,E2 -28362.34} C_VEL
LIN {X 0,Y 65.338,Z 317.158,A -85,B 0,C 180,E1 -28368.814,E2 -28368.814} C_VEL
LIN {X 0,Y 65.206,Z 317.174,A -85,B 0,C 180,E1 -28375.527,E2 -28375.527} C_VEL
LIN {X 0,Y 65.176,Z 317.17,A -85,B 0,C 180,E1 -28382.613,E2 -28382.613} C_VEL
LIN {X 0,Y 65.212,Z 317.165,A -85,B 0,C 180,E1 -28391.078,E2 -28391.078} C_VEL
LIN {X 0,Y 65.233,Z 317.162,A -85,B 0,C 180,E1 -28399.771,E2 -28399.771} C_VEL
LIN {X 0,Y 65.23,Z 317.163,A -85,B 0,C 180,E1 -28409.512,E2 -28409.512} C_VEL
LIN {X 0,Y 65.215,Z 317.172,A -85,B 0,C 180,E1 -28414.501,E2 -28414.501} C_VEL
LIN {X 0,Y 65.568,Z 317.124,A -85,B 0,C 180,E1 -28424.684,E2 -28424.684} C_VEL
LIN {X 0,Y 65.702,Z 317.105,A -85,B 0,C 180,E1 -28427.679,E2 -28427.679} C_VEL
LIN {X 0,Y 66.429,Z 317.023,A -85,B 0,C 180,E1 -28440.03,E2 -28440.03} C_VEL
LIN {X 0,Y 65.713,Z 317.103,A -85,B 0,C 180,E1 -28452.382,E2 -28452.382} C_VEL
LIN {X 0,Y 65.325,Z 317.16,A -85,B 0,C 180,E1 -28458.861,E2 -28458.861} C_VEL
LIN {X 0,Y 65.188,Z 317.176,A -85,B 0,C 180,E1 -28465.579,E2 -28465.579} C_VEL
LIN {X 0,Y 65.155,Z 317.173,A -85,B 0,C 180,E1 -28472.673,E2 -28472.673} C_VEL
LIN {X 0,Y 65.188,Z 317.167,A -85,B 0,C 180,E1 -28481.019,E2 -28481.019} C_VEL
LIN {X 0,Y 65.217,Z 317.164,A -85,B 0,C 180,E1 -28489.73,E2 -28489.73} C_VEL
LIN {X 0,Y 65.333,Z 317.15,A -85,B 0,C 180,E1 -28499.436,E2 -28499.436} C_VEL
LIN {X 0,Y 65.296,Z 317.163,A -85,B 0,C 180,E1 -28504.511,E2 -28504.511} C_VEL
LIN {X 0,Y 67.535,Z 316.879,A -85,B 0,C 180,E1 -28524.037,E2 -28524.037} C_VEL
LIN {X 0,Y 72.103,Z 316.311,A -85,B 0,C 180,E1 -28532.803,E2 -28532.803} C_VEL
LIN {X 0,Y 72.727,Z 316.282,A -85,B 0,C 180,E1 -28533.472,E2 -28533.472} C_VEL
LIN {X 0,Y 76.015,Z 338.211,A -85,B 0,C 180,E1 -28537.064,E2 -28537.064} C_VEL
LIN {X 0,Y 78.285,Z 350.926,A -85,B 0,C 180,E1 -28538.916,E2 -28538.916} C_VEL
LIN {X 0,Y 82.132,Z 381.54,A -85,B 0,C 180,E1 -28544.883,E2 -28544.883} C_VEL
LIN {X 0,Y 83.53,Z 392.164,A -85,B 0,C 180,E1 -28547.766,E2 -28547.766} C_VEL
LIN {X 0,Y 84.818,Z 400.11,A -85,B 0,C 180,E1 -28550.627,E2 -28550.627} C_VEL
LIN {X 0,Y 85.043,Z 402.447,A -85,B 0,C 180,E1 -28551.84,E2 -28551.84} C_VEL
LIN {X 0,Y 85.764,Z 411.779,A -85,B 0,C 180,E1 -28559.459,E2 -28559.459} C_VEL
LIN {X 0,Y 88.583,Z 419.966,A -85,B 0,C 180,E1 -28566.807,E2 -28566.807} C_VEL
LIN {X 0,Y 92.932,Z 426.616,A -85,B 0,C 180,E1 -28572.902,E2 -28572.902} C_VEL
LIN {X 0,Y 94.412,Z 428.311,A -85,B 0,C 180,E1 -28575.623,E2 -28575.623} C_VEL
LIN {X 0,Y 89.322,Z 420.629,A -85,B 0,C 180,E1 -28580.964,E2 -28580.964} C_VEL
LIN {X 0,Y 84.767,Z 410.05,A -85,B 0,C 180,E1 -28588.332,E2 -28588.332} C_VEL
LIN {X 0,Y 82.848,Z 399.795,A -85,B 0,C 180,E1 -28594.878,E2 -28594.878} C_VEL
LIN {X 0,Y 82.076,Z 392.704,A -85,B 0,C 180,E1 -28598.634,E2 -28598.634} C_VEL
LIN {X 0,Y 81.356,Z 385.37,A -85,B 0,C 180,E1 -28601.575,E2 -28601.575} C_VEL
LIN {X 0,Y 80.486,Z 373.425,A -85,B 0,C 180,E1 -28604.967,E2 -28604.967} C_VEL
LIN {X 0,Y 79.29,Z 360.964,A -85,B 0,C 180,E1 -28607.725,E2 -28607.725} C_VEL
LIN {X 0,Y 74.966,Z 320.489,A -85,B 0,C 180,E1 -28615.773,E2 -28615.773} C_VEL
LIN {X 0,Y 74.158,Z 316.056,A -85,B 0,C 180,E1 -28616.407,E2 -28616.407} C_VEL
LIN {X 0,Y 70.322,Z 316.536,A -85,B 0,C 180,E1 -28621.718,E2 -28621.718} C_VEL
LIN {X 0,Y 65.709,Z 317.112,A -85,B 0,C 180,E1 -28638.682,E2 -28638.682} C_VEL
LIN {X 0,Y 65.214,Z 317.165,A -85,B 0,C 180,E1 -28650.423,E2 -28650.423} C_VEL
LIN {X 0,Y 65.161,Z 317.171,A -85,B 0,C 180,E1 -28660.961,E2 -28660.961} C_VEL
LIN {X 0,Y 65.176,Z 317.169,A -85,B 0,C 180,E1 -28669.672,E2 -28669.672} C_VEL
LIN {X 0,Y 65.196,Z 317.167,A -85,B 0,C 180,E1 -28679.518,E2 -28679.518} C_VEL
LIN {X 0,Y 65.166,Z 317.165,A -85,B 0,C 180,E1 -28688.047,E2 -28688.047} C_VEL
LIN {X 0,Y 65.583,Z 317.122,A -85,B 0,C 180,E1 -28694.551,E2 -28694.551} C_VEL
LIN {X 0,Y 65.722,Z 317.102,A -85,B 0,C 180,E1 -28697.64,E2 -28697.64} C_VEL
LIN {X 0,Y 66.463,Z 317.019,A -85,B 0,C 180,E1 -28709.99,E2 -28709.99} C_VEL
LIN {X 0,Y 65.999,Z 317.061,A -85,B 0,C 180,E1 -28713.987,E2 -28713.987} C_VEL
LIN {X 0,Y 65.05,Z 317.195,A -85,B 0,C 180,E1 -28719.083,E2 -28719.083} C_VEL
LIN {X 0,Y 63.349,Z 317.409,A -85,B 0,C 180,E1 -28724.174,E2 -28724.174} C_VEL
LIN {X 0,Y 59.486,Z 317.89,A -85,B 0,C 180,E1 -28734.963,E2 -28734.963} C_VEL
LIN {X 0,Y 58.099,Z 318.049,A -85,B 0,C 180,E1 -28742.841,E2 -28742.841} C_VEL
LIN {X 0,Y 58.058,Z 318.063,A -85,B 0,C 180,E1 -28753.476,E2 -28753.476} C_VEL
LIN {X 0,Y 58.042,Z 318.066,A -85,B 0,C 180,E1 -28762.787,E2 -28762.787} C_VEL
LIN {X 0,Y 58.127,Z 318.054,A -85,B 0,C 180,E1 -28771.119,E2 -28771.119} C_VEL
LIN {X 0,Y 58.443,Z 318.014,A -85,B 0,C 180,E1 -28784.117,E2 -28784.117} C_VEL
LIN {X 0,Y 58.756,Z 317.974,A -85,B 0,C 180,E1 -28793.165,E2 -28793.165} C_VEL
LIN {X 0,Y 59.322,Z 317.908,A -85,B 0,C 180,E1 -28800.034,E2 -28800.034} C_VEL
LIN {X 0,Y 58.76,Z 317.974,A -85,B 0,C 180,E1 -28806.904,E2 -28806.904} C_VEL
LIN {X 0,Y 58.449,Z 318.012,A -85,B 0,C 180,E1 -28815.906,E2 -28815.906} C_VEL
LIN {X 0,Y 58.141,Z 318.046,A -85,B 0,C 180,E1 -28821.298,E2 -28821.298} C_VEL
LIN {X 0,Y 58.112,Z 318.049,A -85,B 0,C 180,E1 -28832.183,E2 -28832.183} C_VEL
LIN {X 0,Y 58.022,Z 318.068,A -85,B 0,C 180,E1 -28837.315,E2 -28837.315} C_VEL
LIN {X 0,Y 58.023,Z 318.067,A -85,B 0,C 180,E1 -28846.661,E2 -28846.661} C_VEL
LIN {X 0,Y 58.219,Z 318.036,A -85,B 0,C 180,E1 -28857.733,E2 -28857.733} C_VEL
LIN {X 0,Y 58.219,Z 318.042,A -85,B 0,C 180,E1 -28861.141,E2 -28861.141} C_VEL
LIN {X 0,Y 58.193,Z 318.041,A -85,B 0,C 180,E1 -28868.771,E2 -28868.771} C_VEL
LIN {X 0,Y 62.553,Z 317.502,A -85,B 0,C 180,E1 -28890.011,E2 -28890.011} C_VEL
LIN {X 0,Y 67.546,Z 316.877,A -85,B 0,C 180,E1 -28897.483,E2 -28897.483} C_VEL
LIN {X 0,Y 67.763,Z 316.851,A -85,B 0,C 180,E1 -28897.646,E2 -28897.646} C_VEL
LIN {X 0,Y 71.211,Z 337.57,A -85,B 0,C 180,E1 -28901.123,E2 -28901.123} C_VEL
LIN {X 0,Y 73.692,Z 350.44,A -85,B 0,C 180,E1 -28902.98,E2 -28902.98} C_VEL
LIN {X 0,Y 78.012,Z 380.366,A -85,B 0,C 180,E1 -28908.931,E2 -28908.931} C_VEL
LIN {X 0,Y 79.384,Z 389.517,A -85,B 0,C 180,E1 -28911.428,E2 -28911.428} C_VEL
LIN {X 0,Y 80.96,Z 397.603,A -85,B 0,C 180,E1 -28914.361,E2 -28914.361} C_VEL
LIN {X 0,Y 81.331,Z 402.868,A -85,B 0,C 180,E1 -28918.389,E2 -28918.389} C_VEL
LIN {X 0,Y 83.358,Z 411.731,A -85,B 0,C 180,E1 -28926.179,E2 -28926.179} C_VEL
LIN {X 0,Y 88.313,Z 420.564,A -85,B 0,C 180,E1 -28934.227,E2 -28934.227} C_VEL
LIN {X 0,Y 87.777,Z 419.777,A -85,B 0,C 180,E1 -28935.74,E2 -28935.74} C_VEL
LIN {X 0,Y 82.193,Z 408.796,A -85,B 0,C 180,E1 -28943.206,E2 -28943.206} C_VEL
LIN {X 0,Y 79.567,Z 399.516,A -85,B 0,C 180,E1 -28949.449,E2 -28949.449} C_VEL
LIN {X 0,Y 78.447,Z 391.656,A -85,B 0,C 180,E1 -28954.004,E2 -28954.004} C_VEL
LIN {X 0,Y 77.489,Z 383.499,A -85,B 0,C 180,E1 -28957.476,E2 -28957.476} C_VEL
LIN {X 0,Y 76.324,Z 372.392,A -85,B 0,C 180,E1 -28960.825,E2 -28960.825} C_VEL
LIN {X 0,Y 74.784,Z 359.998,A -85,B 0,C 180,E1 -28963.718,E2 -28963.718} C_VEL
LIN {X 0,Y 69.776,Z 320.108,A -85,B 0,C 180,E1 -28971.919,E2 -28971.919} C_VEL
LIN {X 0,Y 69.052,Z 316.696,A -85,B 0,C 180,E1 -28972.478,E2 -28972.478} C_VEL
LIN {X 0,Y 63.266,Z 317.417,A -85,B 0,C 180,E1 -28980.522,E2 -28980.522} C_VEL
LIN {X 0,Y 58.395,Z 318.015,A -85,B 0,C 180,E1 -29001.127,E2 -29001.127} C_VEL
LIN {X 0,Y 58.122,Z 318.047,A -85,B 0,C 180,E1 -29012.154,E2 -29012.154} C_VEL
LIN {X 0,Y 58.006,Z 318.071,A -85,B 0,C 180,E1 -29017.24,E2 -29017.24} C_VEL
LIN {X 0,Y 57.987,Z 318.072,A -85,B 0,C 180,E1 -29026.597,E2 -29026.597} C_VEL
LIN {X 0,Y 57.996,Z 318.072,A -85,B 0,C 180,E1 -29032.692,E2 -29032.692} C_VEL
LIN {X 0,Y 58.101,Z 318.057,A -85,B 0,C 180,E1 -29041.05,E2 -29041.05} C_VEL
LIN {X 0,Y 58.477,Z 318.01,A -85,B 0,C 180,E1 -29053.909,E2 -29053.909} C_VEL
LIN {X 0,Y 58.772,Z 317.972,A -85,B 0,C 180,E1 -29063.12,E2 -29063.12} C_VEL
LIN {X 0,Y 59.354,Z 317.905,A -85,B 0,C 180,E1 -29069.989,E2 -29069.989} C_VEL
LIN {X 0,Y 58.768,Z 317.972,A -85,B 0,C 180,E1 -29076.857,E2 -29076.857} C_VEL
LIN {X 0,Y 58.476,Z 318.01,A -85,B 0,C 180,E1 -29086.088,E2 -29086.088} C_VEL
LIN {X 0,Y 58.117,Z 318.055,A -85,B 0,C 180,E1 -29098.914,E2 -29098.914} C_VEL
LIN {X 0,Y 58.099,Z 318.049,A -85,B 0,C 180,E1 -29102.841,E2 -29102.841} C_VEL
LIN {X 0,Y 57.629,Z 318.119,A -85,B 0,C 180,E1 -29106.719,E2 -29106.719} C_VEL
LIN {X 0,Y 56.221,Z 318.289,A -85,B 0,C 180,E1 -29112.529,E2 -29112.529} C_VEL
LIN {X 0,Y 54.412,Z 318.529,A -85,B 0,C 180,E1 -29118.436,E2 -29118.436} C_VEL
LIN {X 0,Y 50.984,Z 318.937,A -85,B 0,C 180,E1 -29136.019,E2 -29136.019} C_VEL
LIN {X 0,Y 51.389,Z 318.891,A -85,B 0,C 180,E1 -29144.168,E2 -29144.168} C_VEL
LIN {X 0,Y 51.633,Z 318.864,A -85,B 0,C 180,E1 -29152.217,E2 -29152.217} C_VEL
LIN {X 0,Y 52.208,Z 318.795,A -85,B 0,C 180,E1 -29160.039,E2 -29160.039} C_VEL
LIN {X 0,Y 51.637,Z 318.864,A -85,B 0,C 180,E1 -29167.862,E2 -29167.862} C_VEL
LIN {X 0,Y 51.311,Z 318.904,A -85,B 0,C 180,E1 -29176.556,E2 -29176.556} C_VEL
LIN {X 0,Y 50.977,Z 318.941,A -85,B 0,C 180,E1 -29184.473,E2 -29184.473} C_VEL
LIN {X 0,Y 50.998,Z 318.941,A -85,B 0,C 180,E1 -29194.248,E2 -29194.248} C_VEL
LIN {X 0,Y 50.987,Z 318.944,A -85,B 0,C 180,E1 -29203.618,E2 -29203.618} C_VEL
LIN {X 0,Y 51.078,Z 318.932,A -85,B 0,C 180,E1 -29215.711,E2 -29215.711} C_VEL
LIN {X 0,Y 51.056,Z 318.931,A -85,B 0,C 180,E1 -29225.624,E2 -29225.624} C_VEL
LIN {X 0,Y 54.914,Z 318.455,A -85,B 0,C 180,E1 -29250.012,E2 -29250.012} C_VEL
LIN {X 0,Y 60.703,Z 317.729,A -85,B 0,C 180,E1 -29260.012,E2 -29260.012} C_VEL
LIN {X 0,Y 63.265,Z 317.4,A -85,B 0,C 180,E1 -29262.542,E2 -29262.542} C_VEL
LIN {X 0,Y 67.684,Z 341,A -85,B 0,C 180,E1 -29266.315,E2 -29266.315} C_VEL
LIN {X 0,Y 69.587,Z 350.216,A -85,B 0,C 180,E1 -29267.647,E2 -29267.647} C_VEL
LIN {X 0,Y 74.569,Z 379.285,A -85,B 0,C 180,E1 -29273.516,E2 -29273.516} C_VEL
LIN {X 0,Y 76.524,Z 389.967,A -85,B 0,C 180,E1 -29276.584,E2 -29276.584} C_VEL
LIN {X 0,Y 77.496,Z 394.661,A -85,B 0,C 180,E1 -29278.443,E2 -29278.443} C_VEL
LIN {X 0,Y 78.848,Z 403.255,A -85,B 0,C 180,E1 -29285.73,E2 -29285.73} C_VEL
LIN {X 0,Y 82.765,Z 412.126,A -85,B 0,C 180,E1 -29293.809,E2 -29293.809} C_VEL
LIN {X 0,Y 82.395,Z 411.529,A -85,B 0,C 180,E1 -29295.09,E2 -29295.09} C_VEL
LIN {X 0,Y 77.771,Z 400.788,A -85,B 0,C 180,E1 -29302.383,E2 -29302.383} C_VEL
LIN {X 0,Y 75.484,Z 391.368,A -85,B 0,C 180,E1 -29308.388,E2 -29308.388} C_VEL
LIN {X 0,Y 74.662,Z 386.221,A -85,B 0,C 180,E1 -29311.127,E2 -29311.127} C_VEL
LIN {X 0,Y 73.548,Z 377.665,A -85,B 0,C 180,E1 -29314.326,E2 -29314.326} C_VEL
LIN {X 0,Y 71.89,Z 364.94,A -85,B 0,C 180,E1 -29317.823,E2 -29317.823} C_VEL
LIN {X 0,Y 65.483,Z 322.916,A -85,B 0,C 180,E1 -29326.79,E2 -29326.79} C_VEL
LIN {X 0,Y 64.43,Z 317.265,A -85,B 0,C 180,E1 -29327.888,E2 -29327.888} C_VEL
LIN {X 0,Y 59.68,Z 317.86,A -85,B 0,C 180,E1 -29333.203,E2 -29333.203} C_VEL
LIN {X 0,Y 55.856,Z 318.34,A -85,B 0,C 180,E1 -29339.964,E2 -29339.964} C_VEL
LIN {X 0,Y 51.638,Z 318.866,A -85,B 0,C 180,E1 -29357.65,E2 -29357.65} C_VEL
LIN {X 0,Y 51.117,Z 318.923,A -85,B 0,C 180,E1 -29364.315,E2 -29364.315} C_VEL
LIN {X 0,Y 50.998,Z 318.941,A -85,B 0,C 180,E1 -29374.2,E2 -29374.2} C_VEL
LIN {X 0,Y 50.954,Z 318.948,A -85,B 0,C 180,E1 -29386.381,E2 -29386.381} C_VEL
LIN {X 0,Y 50.985,Z 318.94,A -85,B 0,C 180,E1 -29396.523,E2 -29396.523} C_VEL
LIN {X 0,Y 50.982,Z 318.94,A -85,B 0,C 180,E1 -29405.557,E2 -29405.557} C_VEL
LIN {X 0,Y 51.425,Z 318.886,A -85,B 0,C 180,E1 -29414.124,E2 -29414.124} C_VEL
LIN {X 0,Y 51.645,Z 318.863,A -85,B 0,C 180,E1 -29422.166,E2 -29422.166} C_VEL
LIN {X 0,Y 52.237,Z 318.791,A -85,B 0,C 180,E1 -29429.987,E2 -29429.987} C_VEL
LIN {X 0,Y 51.643,Z 318.863,A -85,B 0,C 180,E1 -29437.808,E2 -29437.808} C_VEL
LIN {X 0,Y 51.347,Z 318.9,A -85,B 0,C 180,E1 -29446.791,E2 -29446.791} C_VEL
LIN {X 0,Y 50.986,Z 318.939,A -85,B 0,C 180,E1 -29454.411,E2 -29454.411} C_VEL
LIN {X 0,Y 51.014,Z 318.94,A -85,B 0,C 180,E1 -29464.324,E2 -29464.324} C_VEL
LIN {X 0,Y 51.023,Z 318.939,A -85,B 0,C 180,E1 -29473.509,E2 -29473.509} C_VEL
LIN {X 0,Y 51.024,Z 318.939,A -85,B 0,C 180,E1 -29476.53,E2 -29476.53} C_VEL
LIN {X 0,Y 51.043,Z 318.932,A -85,B 0,C 180,E1 -29486.631,E2 -29486.631} C_VEL
LIN {X 0,Y 50.984,Z 318.937,A -85,B 0,C 180,E1 -29496.019,E2 -29496.019} C_VEL
LIN {X 0,Y 50.47,Z 319.008,A -85,B 0,C 180,E1 -29500.431,E2 -29500.431} C_VEL
LIN {X 0,Y 49.327,Z 319.152,A -85,B 0,C 180,E1 -29504.805,E2 -29504.805} C_VEL
LIN {X 0,Y 45.009,Z 319.687,A -85,B 0,C 180,E1 -29520.644,E2 -29520.644} C_VEL
LIN {X 0,Y 44.479,Z 319.757,A -85,B 0,C 180,E1 -29529.137,E2 -29529.137} C_VEL
LIN {X 0,Y 44.071,Z 319.807,A -85,B 0,C 180,E1 -29538.646,E2 -29538.646} C_VEL
LIN {X 0,Y 43.797,Z 319.837,A -85,B 0,C 180,E1 -29548.828,E2 -29548.828} C_VEL
LIN {X 0,Y 43.825,Z 319.838,A -85,B 0,C 180,E1 -29556.722,E2 -29556.722} C_VEL
LIN {X 0,Y 43.825,Z 319.828,A -85,B 0,C 180,E1 -29570.12,E2 -29570.12} C_VEL
LIN {X 0,Y 43.877,Z 319.832,A -85,B 0,C 180,E1 -29573.286,E2 -29573.286} C_VEL
LIN {X 0,Y 43.885,Z 319.827,A -85,B 0,C 180,E1 -29581.304,E2 -29581.304} C_VEL
LIN {X 0,Y 44.189,Z 319.793,A -85,B 0,C 180,E1 -29592.747,E2 -29592.747} C_VEL
LIN {X 0,Y 50.771,Z 318.97,A -85,B 0,C 180,E1 -29617.97,E2 -29617.97} C_VEL
LIN {X 0,Y 55.482,Z 318.375,A -85,B 0,C 180,E1 -29624.688,E2 -29624.688} C_VEL
LIN {X 0,Y 59.443,Z 317.901,A -85,B 0,C 180,E1 -29628.205,E2 -29628.205} C_VEL
LIN {X 0,Y 64.694,Z 342.89,A -85,B 0,C 180,E1 -29631.938,E2 -29631.938} C_VEL
LIN {X 0,Y 66.155,Z 349.562,A -85,B 0,C 180,E1 -29632.867,E2 -29632.867} C_VEL
LIN {X 0,Y 71.729,Z 378.315,A -85,B 0,C 180,E1 -29638.542,E2 -29638.542} C_VEL
LIN {X 0,Y 73.978,Z 389.179,A -85,B 0,C 180,E1 -29641.725,E2 -29641.725} C_VEL
LIN {X 0,Y 74.232,Z 390.167,A -85,B 0,C 180,E1 -29642.091,E2 -29642.091} C_VEL
LIN {X 0,Y 74.75,Z 393.233,A -85,B 0,C 180,E1 -29644.352,E2 -29644.352} C_VEL
LIN {X 0,Y 77.631,Z 402.644,A -85,B 0,C 180,E1 -29652.779,E2 -29652.779} C_VEL
LIN {X 0,Y 78.051,Z 403.559,A -85,B 0,C 180,E1 -29653.883,E2 -29653.883} C_VEL
LIN {X 0,Y 74.005,Z 392.923,A -85,B 0,C 180,E1 -29660.98,E2 -29660.98} C_VEL
LIN {X 0,Y 72.115,Z 384.303,A -85,B 0,C 180,E1 -29666.097,E2 -29666.097} C_VEL
LIN {X 0,Y 70.664,Z 376.044,A -85,B 0,C 180,E1 -29669.324,E2 -29669.324} C_VEL
LIN {X 0,Y 68.721,Z 364.237,A -85,B 0,C 180,E1 -29672.628,E2 -29672.628} C_VEL
LIN {X 0,Y 62.31,Z 327.972,A -85,B 0,C 180,E1 -29680.332,E2 -29680.332} C_VEL
LIN {X 0,Y 60.563,Z 317.851,A -85,B 0,C 180,E1 -29682.383,E2 -29682.383} C_VEL
LIN {X 0,Y 56.728,Z 318.224,A -85,B 0,C 180,E1 -29685.618,E2 -29685.618} C_VEL
LIN {X 0,Y 48.225,Z 319.291,A -85,B 0,C 180,E1 -29699.958,E2 -29699.958} C_VEL
LIN {X 0,Y 44.448,Z 319.761,A -85,B 0,C 180,E1 -29718.386,E2 -29718.386} C_VEL
LIN {X 0,Y 43.858,Z 319.83,A -85,B 0,C 180,E1 -29728.679,E2 -29728.679} C_VEL
LIN {X 0,Y 43.776,Z 319.834,A -85,B 0,C 180,E1 -29739.891,E2 -29739.891} C_VEL
LIN {X 0,Y 43.804,Z 319.84,A -85,B 0,C 180,E1 -29753.26,E2 -29753.26} C_VEL
LIN {X 0,Y 43.79,Z 319.838,A -85,B 0,C 180,E1 -29761.201,E2 -29761.201} C_VEL
LIN {X 0,Y 44.196,Z 319.792,A -85,B 0,C 180,E1 -29772.414,E2 -29772.414} C_VEL
LIN {X 0,Y 44.498,Z 319.755,A -85,B 0,C 180,E1 -29780.897,E2 -29780.897} C_VEL
LIN {X 0,Y 45.111,Z 319.679,A -85,B 0,C 180,E1 -29789.985,E2 -29789.985} C_VEL
LIN {X 0,Y 44.494,Z 319.755,A -85,B 0,C 180,E1 -29799.072,E2 -29799.072} C_VEL
LIN {X 0,Y 44.114,Z 319.802,A -85,B 0,C 180,E1 -29808.564,E2 -29808.564} C_VEL
LIN {X 0,Y 43.816,Z 319.835,A -85,B 0,C 180,E1 -29818.745,E2 -29818.745} C_VEL
LIN {X 0,Y 43.832,Z 319.827,A -85,B 0,C 180,E1 -29829.872,E2 -29829.872} C_VEL
LIN {X 0,Y 43.858,Z 319.834,A -85,B 0,C 180,E1 -29843.221,E2 -29843.221} C_VEL
LIN {X 0,Y 43.823,Z 319.834,A -85,B 0,C 180,E1 -29851.296,E2 -29851.296} C_VEL
LIN {X 0,Y 44.17,Z 319.795,A -85,B 0,C 180,E1 -29862.629,E2 -29862.629} C_VEL
LIN {X 0,Y 44.482,Z 319.757,A -85,B 0,C 180,E1 -29870.956,E2 -29870.956} C_VEL
LIN {X 0,Y 45.009,Z 319.687,A -85,B 0,C 180,E1 -29880.644,E2 -29880.644} C_VEL
LIN {X 0,Y 44.171,Z 319.785,A -85,B 0,C 180,E1 -29885.6,E2 -29885.6} C_VEL
LIN {X 0,Y 42.326,Z 320.022,A -85,B 0,C 180,E1 -29893.089,E2 -29893.089} C_VEL
LIN {X 0,Y 40.207,Z 320.28,A -85,B 0,C 180,E1 -29900.868,E2 -29900.868} C_VEL
LIN {X 0,Y 36.596,Z 320.711,A -85,B 0,C 180,E1 -29925.116,E2 -29925.116} C_VEL
LIN {X 0,Y 36.744,Z 320.709,A -85,B 0,C 180,E1 -29929.996,E2 -29929.996} C_VEL
LIN {X 0,Y 36.757,Z 320.716,A -85,B 0,C 180,E1 -29935.021,E2 -29935.021} C_VEL
LIN {X 0,Y 37.041,Z 320.684,A -85,B 0,C 180,E1 -29951.73,E2 -29951.73} C_VEL
LIN {X 0,Y 43.163,Z 319.92,A -85,B 0,C 180,E1 -29979.387,E2 -29979.387} C_VEL
LIN {X 0,Y 47.947,Z 319.324,A -85,B 0,C 180,E1 -29987.062,E2 -29987.062} C_VEL
LIN {X 0,Y 56.289,Z 318.28,A -85,B 0,C 180,E1 -29994.566,E2 -29994.566} C_VEL
LIN {X 0,Y 62.129,Z 343.702,A -85,B 0,C 180,E1 -29997.919,E2 -29997.919} C_VEL
LIN {X 0,Y 63.507,Z 349.706,A -85,B 0,C 180,E1 -29998.743,E2 -29998.743} C_VEL
LIN {X 0,Y 69.574,Z 377.344,A -85,B 0,C 180,E1 -30003.98,E2 -30003.98} C_VEL
LIN {X 0,Y 71.889,Z 387.016,A -85,B 0,C 180,E1 -30006.806,E2 -30006.806} C_VEL
LIN {X 0,Y 73.494,Z 393.057,A -85,B 0,C 180,E1 -30012.031,E2 -30012.031} C_VEL
LIN {X 0,Y 73.709,Z 393.818,A -85,B 0,C 180,E1 -30013.457,E2 -30013.457} C_VEL
LIN {X 0,Y 70.748,Z 384.705,A -85,B 0,C 180,E1 -30019.28,E2 -30019.28} C_VEL
LIN {X 0,Y 69.439,Z 378.725,A -85,B 0,C 180,E1 -30022.345,E2 -30022.345} C_VEL
LIN {X 0,Y 67.396,Z 368.426,A -85,B 0,C 180,E1 -30025.707,E2 -30025.707} C_VEL
LIN {X 0,Y 64.813,Z 356.193,A -85,B 0,C 180,E1 -30028.509,E2 -30028.509} C_VEL
LIN {X 0,Y 57.452,Z 319.23,A -85,B 0,C 180,E1 -30036.178,E2 -30036.178} C_VEL
LIN {X 0,Y 57.071,Z 318.18,A -85,B 0,C 180,E1 -30036.371,E2 -30036.371} C_VEL
LIN {X 0,Y 52.465,Z 318.759,A -85,B 0,C 180,E1 -30039.704,E2 -30039.704} C_VEL
LIN {X 0,Y 42.355,Z 320.012,A -85,B 0,C 180,E1 -30054.778,E2 -30054.778} C_VEL
LIN {X 0,Y 37.241,Z 320.655,A -85,B 0,C 180,E1 -30079.283,E2 -30079.283} C_VEL
LIN {X 0,Y 36.706,Z 320.722,A -85,B 0,C 180,E1 -30094.989,E2 -30094.989} C_VEL
LIN {X 0,Y 36.699,Z 320.715,A -85,B 0,C 180,E1 -30099.975,E2 -30099.975} C_VEL
LIN {X 0,Y 36.693,Z 320.716,A -85,B 0,C 180,E1 -30109.919,E2 -30109.919} C_VEL
LIN {X 0,Y 36.682,Z 320.726,A -85,B 0,C 180,E1 -30114.894,E2 -30114.894} C_VEL
LIN {X 0,Y 37.022,Z 320.685,A -85,B 0,C 180,E1 -30131.471,E2 -30131.471} C_VEL
LIN {X 0,Y 37.294,Z 320.645,A -85,B 0,C 180,E1 -30139.119,E2 -30139.119} C_VEL
LIN {X 0,Y 37.968,Z 320.568,A -85,B 0,C 180,E1 -30149.982,E2 -30149.982} C_VEL
LIN {X 0,Y 37.29,Z 320.646,A -85,B 0,C 180,E1 -30160.845,E2 -30160.845} C_VEL
LIN {X 0,Y 37.017,Z 320.686,A -85,B 0,C 180,E1 -30168.507,E2 -30168.507} C_VEL
LIN {X 0,Y 36.718,Z 320.721,A -85,B 0,C 180,E1 -30185.021,E2 -30185.021} C_VEL
LIN {X 0,Y 36.743,Z 320.709,A -85,B 0,C 180,E1 -30190.173,E2 -30190.173} C_VEL
LIN {X 0,Y 36.746,Z 320.709,A -85,B 0,C 180,E1 -30199.881,E2 -30199.881} C_VEL
LIN {X 0,Y 36.723,Z 320.72,A -85,B 0,C 180,E1 -30205.031,E2 -30205.031} C_VEL
LIN {X 0,Y 37.009,Z 320.688,A -85,B 0,C 180,E1 -30221.653,E2 -30221.653} C_VEL
LIN {X 0,Y 37.279,Z 320.648,A -85,B 0,C 180,E1 -30229.189,E2 -30229.189} C_VEL
LIN {X 0,Y 37.943,Z 320.572,A -85,B 0,C 180,E1 -30240.053,E2 -30240.053} C_VEL
LIN {X 0,Y 37.257,Z 320.65,A -85,B 0,C 180,E1 -30250.928,E2 -30250.928} C_VEL
LIN {X 0,Y 37.008,Z 320.688,A -85,B 0,C 180,E1 -30258.343,E2 -30258.343} C_VEL
LIN {X 0,Y 36.701,Z 320.724,A -85,B 0,C 180,E1 -30275.128,E2 -30275.128} C_VEL
LIN {X 0,Y 36.722,Z 320.712,A -85,B 0,C 180,E1 -30280.076,E2 -30280.076} C_VEL
LIN {X 0,Y 36.596,Z 320.711,A -85,B 0,C 180,E1 -30285.116,E2 -30285.116} C_VEL
LIN {X 0,Y 36.255,Z 320.772,A -85,B 0,C 180,E1 -30291.198,E2 -30291.198} C_VEL
LIN {X 0,Y 34.918,Z 320.943,A -85,B 0,C 180,E1 -30300.433,E2 -30300.433} C_VEL
LIN {X 0,Y 32.605,Z 321.197,A -85,B 0,C 180,E1 -30317.225,E2 -30317.225} C_VEL
LIN {X 0,Y 33.25,Z 321.132,A -85,B 0,C 180,E1 -30333.415,E2 -30333.415} C_VEL
LIN {X 0,Y 34.496,Z 320.962,A -85,B 0,C 180,E1 -30338.188,E2 -30338.188} C_VEL
LIN {X 0,Y 40.566,Z 320.238,A -85,B 0,C 180,E1 -30350.291,E2 -30350.291} C_VEL
LIN {X 0,Y 47.684,Z 319.358,A -85,B 0,C 180,E1 -30357.746,E2 -30357.746} C_VEL
LIN {X 0,Y 54.068,Z 318.55,A -85,B 0,C 180,E1 -30361.597,E2 -30361.597} C_VEL
LIN {X 0,Y 60.237,Z 343.536,A -85,B 0,C 180,E1 -30364.318,E2 -30364.318} C_VEL
LIN {X 0,Y 61.757,Z 349.729,A -85,B 0,C 180,E1 -30365.128,E2 -30365.128} C_VEL
LIN {X 0,Y 68.204,Z 376.062,A -85,B 0,C 180,E1 -30369.673,E2 -30369.673} C_VEL
LIN {X 0,Y 70.188,Z 383.564,A -85,B 0,C 180,E1 -30371.76,E2 -30371.76} C_VEL
LIN {X 0,Y 70.318,Z 384.09,A -85,B 0,C 180,E1 -30372.217,E2 -30372.217} C_VEL
LIN {X 0,Y 70.105,Z 383.527,A -85,B 0,C 180,E1 -30372.948,E2 -30372.948} C_VEL
LIN {X 0,Y 68.124,Z 376.829,A -85,B 0,C 180,E1 -30376.688,E2 -30376.688} C_VEL
LIN {X 0,Y 66.252,Z 368.893,A -85,B 0,C 180,E1 -30379.329,E2 -30379.329} C_VEL
LIN {X 0,Y 63.398,Z 356.8,A -85,B 0,C 180,E1 -30382.147,E2 -30382.147} C_VEL
LIN {X 0,Y 54.638,Z 318.482,A -85,B 0,C 180,E1 -30389.53,E2 -30389.53} C_VEL
LIN {X 0,Y 47.678,Z 319.357,A -85,B 0,C 180,E1 -30393.709,E2 -30393.709} C_VEL
LIN {X 0,Y 35.553,Z 320.869,A -85,B 0,C 180,E1 -30411.375,E2 -30411.375} C_VEL
LIN {X 0,Y 30.034,Z 321.434,A -85,B 0,C 180,E1 -30440.545,E2 -30440.545} C_VEL
LIN {X 0,Y 29.589,Z 321.477,A -85,B 0,C 180,E1 -30448.283,E2 -30448.283} C_VEL
LIN {X 0,Y 29.517,Z 321.484,A -85,B 0,C 180,E1 -30465.485,E2 -30465.485} C_VEL
LIN {X 0,Y 29.455,Z 321.489,A -85,B 0,C 180,E1 -30481.472,E2 -30481.472} C_VEL
LIN {X 0,Y 29.827,Z 321.454,A -85,B 0,C 180,E1 -30490.266,E2 -30490.266} C_VEL
LIN {X 0,Y 30.071,Z 321.429,A -85,B 0,C 180,E1 -30496.461,E2 -30496.461} C_VEL
LIN {X 0,Y 30.785,Z 321.366,A -85,B 0,C 180,E1 -30509.978,E2 -30509.978} C_VEL
LIN {X 0,Y 30.067,Z 321.429,A -85,B 0,C 180,E1 -30523.494,E2 -30523.494} C_VEL
LIN {X 0,Y 29.827,Z 321.454,A -85,B 0,C 180,E1 -30529.734,E2 -30529.734} C_VEL
LIN {X 0,Y 29.474,Z 321.488,A -85,B 0,C 180,E1 -30538.456,E2 -30538.456} C_VEL
LIN {X 0,Y 29.564,Z 321.479,A -85,B 0,C 180,E1 -30555.459,E2 -30555.459} C_VEL
LIN {X 0,Y 29.475,Z 321.487,A -85,B 0,C 180,E1 -30571.599,E2 -30571.599} C_VEL
LIN {X 0,Y 29.823,Z 321.455,A -85,B 0,C 180,E1 -30580.43,E2 -30580.43} C_VEL
LIN {X 0,Y 30.06,Z 321.43,A -85,B 0,C 180,E1 -30586.549,E2 -30586.549} C_VEL
LIN {X 0,Y 30.756,Z 321.369,A -85,B 0,C 180,E1 -30600.066,E2 -30600.066} C_VEL
LIN {X 0,Y 30.049,Z 321.431,A -85,B 0,C 180,E1 -30613.594,E2 -30613.594} C_VEL
LIN {X 0,Y 29.819,Z 321.455,A -85,B 0,C 180,E1 -30619.553,E2 -30619.553} C_VEL
LIN {X 0,Y 29.464,Z 321.488,A -85,B 0,C 180,E1 -30628.57,E2 -30628.57} C_VEL
LIN {X 0,Y 29.554,Z 321.481,A -85,B 0,C 180,E1 -30645.608,E2 -30645.608} C_VEL
LIN {X 0,Y 29.516,Z 321.485,A -85,B 0,C 180,E1 -30661.588,E2 -30661.588} C_VEL
LIN {X 0,Y 30.245,Z 321.412,A -85,B 0,C 180,E1 -30676.587,E2 -30676.587} C_VEL
LIN {X 0,Y 34.496,Z 320.962,A -85,B 0,C 180,E1 -30698.188,E2 -30698.188} C_VEL
LIN {X 0,Y 36.12,Z 320.791,A -85,B 0,C 180,E1 -30704.171,E2 -30704.171} C_VEL
LIN {X 0,Y 41.569,Z 320.11,A -85,B 0,C 180,E1 -30722.498,E2 -30722.498} C_VEL
LIN {X 0,Y 44.7,Z 319.723,A -85,B 0,C 180,E1 -30725.633,E2 -30725.633} C_VEL
LIN {X 0,Y 52.921,Z 318.695,A -85,B 0,C 180,E1 -30729.126,E2 -30729.126} C_VEL
LIN {X 0,Y 59.498,Z 344.314,A -85,B 0,C 180,E1 -30731.09,E2 -30731.09} C_VEL
LIN {X 0,Y 64.456,Z 363.329,A -85,B 0,C 180,E1 -30733.81,E2 -30733.81} C_VEL
LIN {X 0,Y 64.494,Z 363.512,A -85,B 0,C 180,E1 -30734.245,E2 -30734.245} C_VEL
LIN {X 0,Y 61.297,Z 351.579,A -85,B 0,C 180,E1 -30736.491,E2 -30736.491} C_VEL
LIN {X 0,Y 53.144,Z 318.67,A -85,B 0,C 180,E1 -30742.122,E2 -30742.122} C_VEL
LIN {X 0,Y 47.894,Z 319.326,A -85,B 0,C 180,E1 -30744.008,E2 -30744.008} C_VEL
LIN {X 0,Y 40.706,Z 320.216,A -85,B 0,C 180,E1 -30748.749,E2 -30748.749} C_VEL
LIN {X 0,Y 28.935,Z 321.536,A -85,B 0,C 180,E1 -30766.397,E2 -30766.397} C_VEL
LIN {X 0,Y 23.054,Z 321.87,A -85,B 0,C 180,E1 -30797.656,E2 -30797.656} C_VEL
LIN {X 0,Y 22.205,Z 321.897,A -85,B 0,C 180,E1 -30819.152,E2 -30819.152} C_VEL
LIN {X 0,Y 22.166,Z 321.898,A -85,B 0,C 180,E1 -30830.607,E2 -30830.607} C_VEL
LIN {X 0,Y 22.77,Z 321.879,A -85,B 0,C 180,E1 -30851.991,E2 -30851.991} C_VEL
LIN {X 0,Y 23.553,Z 321.855,A -85,B 0,C 180,E1 -30869.971,E2 -30869.971} C_VEL
LIN {X 0,Y 22.777,Z 321.879,A -85,B 0,C 180,E1 -30887.941,E2 -30887.941} C_VEL
LIN {X 0,Y 22.19,Z 321.897,A -85,B 0,C 180,E1 -30909.263,E2 -30909.263} C_VEL
LIN {X 0,Y 22.191,Z 321.897,A -85,B 0,C 180,E1 -30920.819,E2 -30920.819} C_VEL
LIN {X 0,Y 22.767,Z 321.879,A -85,B 0,C 180,E1 -30942.114,E2 -30942.114} C_VEL
LIN {X 0,Y 23.527,Z 321.856,A -85,B 0,C 180,E1 -30960.086,E2 -30960.086} C_VEL
LIN {X 0,Y 22.748,Z 321.88,A -85,B 0,C 180,E1 -30978.088,E2 -30978.088} C_VEL
LIN {X 0,Y 22.194,Z 321.897,A -85,B 0,C 180,E1 -30999.412,E2 -30999.412} C_VEL
LIN {X 0,Y 22.21,Z 321.897,A -85,B 0,C 180,E1 -31010.779,E2 -31010.779} C_VEL
LIN {X 0,Y 22.801,Z 321.878,A -85,B 0,C 180,E1 -31032.079,E2 -31032.079} C_VEL
LIN {X 0,Y 29.542,Z 321.483,A -85,B 0,C 180,E1 -31067.686,E2 -31067.686} C_VEL
LIN {X 0,Y 39.751,Z 320.335,A -85,B 0,C 180,E1 -31082.053,E2 -31082.053} C_VEL
LIN {X 0,Y 44.7,Z 319.723,A -85,B 0,C 180,E1 -31085.633,E2 -31085.633} C_VEL
LIN {X 0,Y 45.096,Z 319.676,A -85,B 0,C 180,E1 -31087.245,E2 -31087.245} C_VEL
LIN {X 0,Y 43.93,Z 319.829,A -85,B 0,C 180,E1 -31090.258,E2 -31090.258} C_VEL
LIN {X 0,Y 39.908,Z 320.34,A -85,B 0,C 180,E1 -31095.191,E2 -31095.191} C_VEL
LIN {X 0,Y 33.648,Z 321.091,A -85,B 0,C 180,E1 -31101.085,E2 -31101.085} C_VEL
LIN {X 0,Y 24.518,Z 321.825,A -85,B 0,C 180,E1 -31114.203,E2 -31114.203} C_VEL
LIN {X 0,Y 20.575,Z 321.93,A -85,B 0,C 180,E1 -31124.484,E2 -31124.484} C_VEL
LIN {X 0,Y 17.398,Z 321.991,A -85,B 0,C 180,E1 -31139.884,E2 -31139.884} C_VEL
LIN {X 0,Y 15.221,Z 321.991,A -85,B 0,C 180,E1 -31167.347,E2 -31167.347} C_VEL
LIN {X 0,Y 15.034,Z 321.991,A -85,B 0,C 180,E1 -31202.079,E2 -31202.079} C_VEL
LIN {X 0,Y 15.223,Z 321.991,A -85,B 0,C 180,E1 -31207.066,E2 -31207.066} C_VEL
LIN {X 0,Y 16.218,Z 321.991,A -85,B 0,C 180,E1 -31229.958,E2 -31229.958} C_VEL
LIN {X 0,Y 15.244,Z 321.991,A -85,B 0,C 180,E1 -31253.116,E2 -31253.116} C_VEL
LIN {X 0,Y 15.072,Z 321.991,A -85,B 0,C 180,E1 -31257.742,E2 -31257.742} C_VEL
LIN {X 0,Y 15.073,Z 321.991,A -85,B 0,C 180,E1 -31292.361,E2 -31292.361} C_VEL
LIN {X 0,Y 15.248,Z 321.991,A -85,B 0,C 180,E1 -31297.082,E2 -31297.082} C_VEL
LIN {X 0,Y 16.193,Z 321.991,A -85,B 0,C 180,E1 -31320.125,E2 -31320.125} C_VEL
LIN {X 0,Y 15.235,Z 321.991,A -85,B 0,C 180,E1 -31342.802,E2 -31342.802} C_VEL
LIN {X 0,Y 15.045,Z 321.991,A -85,B 0,C 180,E1 -31347.999,E2 -31347.999} C_VEL
LIN {X 0,Y 15.078,Z 321.991,A -85,B 0,C 180,E1 -31382.27,E2 -31382.27} C_VEL
LIN {X 0,Y 16.927,Z 321.991,A -85,B 0,C 180,E1 -31410.04,E2 -31410.04} C_VEL
LIN {X 0,Y 26.665,Z 321.742,A -85,B 0,C 180,E1 -31441.842,E2 -31441.842} C_VEL
LIN {X 0,Y 40.657,Z 320.231,A -85,B 0,C 180,E1 -31453.767,E2 -31453.767} C_VEL
LIN {X 0,Y 42.034,Z 320.06,A -85,B 0,C 180,E1 -31454.303,E2 -31454.303} C_VEL
LIN {X 0,Y 42.65,Z 319.981,A -85,B 0,C 180,E1 -31456.951,E2 -31456.951} C_VEL
LIN {X 0,Y 34.222,Z 321.027,A -85,B 0,C 180,E1 -31461.896,E2 -31461.896} C_VEL
LIN {X 0,Y 22.696,Z 321.881,A -85,B 0,C 180,E1 -31478.353,E2 -31478.353} C_VEL
LIN {X 0,Y 20.575,Z 321.93,A -85,B 0,C 180,E1 -31484.484,E2 -31484.484} C_VEL
LIN {X 0,Y 17.82,Z 321.993,A -85,B 0,C 180,E1 -31493,E2 -31493} C_VEL
LIN {X 0,Y 14.802,Z 321.993,A -85,B 0,C 180,E1 -31502.251,E2 -31502.251} C_VEL
LIN {X 0,Y 9.144,Z 321.993,A -85,B 0,C 180,E1 -31531.858,E2 -31531.858} C_VEL
LIN {X 0,Y 7.781,Z 321.991,A -85,B 0,C 180,E1 -31569.062,E2 -31569.062} C_VEL
LIN {X 0,Y 8.645,Z 321.991,A -85,B 0,C 180,E1 -31589.921,E2 -31589.921} C_VEL
LIN {X 0,Y 7.744,Z 321.991,A -85,B 0,C 180,E1 -31615.454,E2 -31615.454} C_VEL
LIN {X 0,Y 7.753,Z 321.991,A -85,B 0,C 180,E1 -31654.821,E2 -31654.821} C_VEL
LIN {X 0,Y 8.633,Z 321.991,A -85,B 0,C 180,E1 -31680.234,E2 -31680.234} C_VEL
LIN {X 0,Y 7.756,Z 321.991,A -85,B 0,C 180,E1 -31705.231,E2 -31705.231} C_VEL
LIN {X 0,Y 7.783,Z 321.991,A -85,B 0,C 180,E1 -31745.167,E2 -31745.167} C_VEL
LIN {X 0,Y 9.062,Z 321.991,A -85,B 0,C 180,E1 -31770.075,E2 -31770.075} C_VEL
LIN {X 0,Y 20.533,Z 321.947,A -85,B 0,C 180,E1 -31813.244,E2 -31813.244} C_VEL
LIN {X 0,Y 21.235,Z 321.927,A -85,B 0,C 180,E1 -31818.429,E2 -31818.429} C_VEL
LIN {X 0,Y 9.376,Z 321.991,A -85,B 0,C 180,E1 -31859.784,E2 -31859.784} C_VEL
LIN {X 0,Y 7.814,Z 321.991,A -85,B 0,C 180,E1 -31885.728,E2 -31885.728} C_VEL
LIN {X 0,Y 7.781,Z 321.991,A -85,B 0,C 180,E1 -31929.062,E2 -31929.062} C_VEL
LIN {X 0,Y 7.05,Z 321.991,A -85,B 0,C 180,E1 -31938.065,E2 -31938.065} C_VEL
LIN {X 0,Y 4.807,Z 321.991,A -85,B 0,C 180,E1 -31947.946,E2 -31947.946} C_VEL
LIN {X 0,Y 1.591,Z 321.991,A -85,B 0,C 180,E1 -31973.722,E2 -31973.722} C_VEL
LIN {X 0,Y 0.353,Z 321.991,A -85,B 0,C 180,E1 -32085.538,E2 -32085.538} C_VEL
LIN {X 0,Y 0.3,Z 321.991,A -85,B 0,C 180,E1 -32132.275,E2 -32132.275} C_VEL
LIN {X 0,Y 0.381,Z 321.991,A -85,B 0,C 180,E1 -32214.676,E2 -32214.676} C_VEL
LIN {X 0,Y 0.32,Z 321.991,A -85,B 0,C 180,E1 -32307.87,E2 -32307.87} C_VEL
LIN {X 0,Y 0.254,Z 321.991,A -85,B 0,C 180,E1 -32407.992,E2 -32407.992} C_VEL
LIN {X 0,Y 0.3,Z 321.991,A -85,B 0,C 180,E1 -32492.275,E2 -32492.275} C_VEL
LIN {X 0,Y 2.23,Z 323.991,A -85,B 0,C 180,E1 -32529.706,E2 -32529.706} C_VEL
LIN {X 0,Y 2.23,Z 600,A -85,B 0,C 180,E1 -32529.706,E2 -32529.706} C_VEL
LIN {X 0,Y 2.23,Z 600,A -85,B 0,C 180,E1 -32529.706,E2 -32529.706}

QRS_NEXT_CUT()

QRS_NEXT()
QRS_HOME()

END
